PROGRAM main
  VAR
    HS101A_Green AT %IX0.0 : BOOL; (* Green push button, momentary normally open *)
    HS101B_Yellow AT %IX0.1 : BOOL; (* Yellow push button, momentary, normally open *)
    HS101C_Red AT %IX0.2 : BOOL; (* Red push button, momentary, normally open *)
    XL101A_Green AT %QX0.0 : BOOL; (* Green stoplight *)
    XL101B_Yellow AT %QX0.1 : BOOL; (* Yellow stoplight *)
    XL101C_Red AT %QX0.2 : BOOL; (* Red stoplight *)
  END_VAR

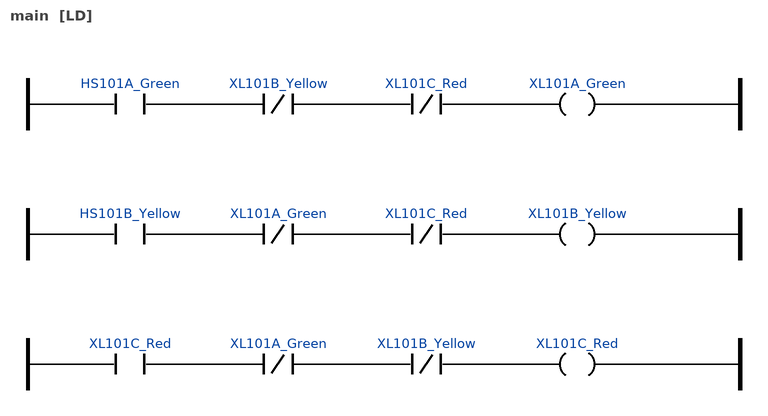
(* LD diagram, written out as Structured Text *)
XL101A_Green := HS101A_Green AND NOT XL101B_Yellow AND NOT XL101C_Red;
XL101B_Yellow := HS101B_Yellow AND NOT XL101A_Green AND NOT XL101C_Red;
XL101C_Red := XL101C_Red AND NOT XL101A_Green AND NOT XL101B_Yellow;
END_PROGRAM
